TYPE ForceLimiterFsmAction :
(
	FsmAction_None := stdNOV.FSM_ACTION_NONE,	
	FsmAction_Warn := 1,
	FsmAction_Crit_Alarm,	
	FsmAction_Clear_Warning,
	FsmAction_Clear_Crit_Alarm,	
	NUM_FsmActions
) BYTE;
END_TYPE

(* stored: Version 1.1.0.1, ProductVersion 3.1.4024.6
   DUT ForceLimiterFsmAction: Id {0ac4eab1-eb97-4604-bf82-0524872cae92} *)
